TYPE DUT_NextPartPLCData :
STRUCT
	return_value: DINT;
	PLCData : STRING(DB.MAX_STRING_SIZE);
END_STRUCT
END_TYPE

(* stored: Version 1.1.0.1, ProductVersion 3.1.4024.15
   DUT DUT_NextPartPLCData: Id {c2ec7f98-dab3-496e-a47b-c1ff79a92ad2} *)
